Fanuc KAREL source: INI_DYN_DISI.kl

PROGRAM T
%NOLOCKGROUP
VAR
 v0 : INTEGER
 v1 : STRING[40]
 v2 : INTEGER
 v3 : INTEGER
 v4 : INTEGER
 v5 : INTEGER
 v6 : INTEGER
 v7 : INTEGER
 v8 : INTEGER
 v9 : STRING[40]
 v10 : INTEGER
BEGIN
 INI_DYN_DISI(v0, v1, v2, v3, v4, v5, v6, v7, v8, v9, v10)
END T
